FUNCTION_BLOCK Outfeed EXTENDS FB_PackML_BaseModule
VAR
	iOutfeedxis				   : I_BasicAxis;				  // For most axis and component commands
	iOutfeedAxisComponent	   : I_ComponentBase;			  // For registering the component with the EM
	iExternalSetpointGenerator : I_ExternalSetpointGenerator; // For setting properties of the External Setpoint Generator
END_VAR

// This method contains code which will execute when this PackML module is in the Aborting state
METHOD PROTECTED Aborting

// Note: The Abort command should be associated with the fault handing routine of a module. It should not be directly commanded from any user inteface. 

// This method is called as required by <c>StateControl()</c>
CASE SequenceState OF
	0:
		NoStateTasksToComplete := FALSE;
		SequenceState		   := SequenceState + 10;

	10:
		IF NOT iOutfeedxis.Error THEN
			IF iOutfeedxis.Stop() THEN
				SequenceState := SequenceState + 10;
			END_IF
		ELSE
			SequenceState := SequenceState + 10;
		END_IF

	20:
		IF iOutfeedxis.Stopped THEN
			SequenceState := SequenceState + 10;
		END_IF

	30:
		IF iOutfeedxis.Disable() THEN
			SequenceState := SequenceState + 10;
		END_IF

	40:
		IF NOT iOutfeedxis.Enabled THEN
			SequenceState := SequenceState + 10;
		END_IF

	50:
		StateTasksComplete := TRUE;
END_CASE

SUPER^.Aborting();
END_METHOD

// This method contains code which will execute when this PackML module is in the Clearing state
METHOD PROTECTED Clearing
VAR
	i				: UDINT;
	SubModulesReady : BOOL := TRUE;
END_VAR

// Note: The Clear command can also be thought of as a fault reset depite the ambiguity in the naming of the Reset state. 

// This method is called as required by <c>StateControl()</c>
CASE SequenceState OF
	0:
		NoStateTasksToComplete := FALSE;
		SequenceState		   := SequenceState + 10;

	10:
		IF iOutfeedxis.Reset() THEN
			SequenceState := SequenceState + 10;
		END_IF

	20:
		IF NOT iOutfeedxis.Error THEN
			SequenceState := SequenceState + 10;
		END_IF

	30:
		StateTasksComplete := TRUE;
END_CASE

SUPER^.Clearing();
END_METHOD

// This method contains code which will execute when this PackML module is in the Execute state
METHOD PROTECTED Execute
VAR
	

END_VAR

(*
The base implementation of this method is empty. User must override this method to provide functionality.
This method is called as required by StateControl()
*)
VAR
	Position : LREAL;
END_VAR
CASE _CurrentMode OF
	E_PMLUnitMode.ePMLUnitMode_Production:
		CASE SequenceState OF
			0:
				iExternalSetpointGenerator.Direction   := 1;
				iExternalSetpointGenerator.Destination := 0.0;
				iExternalSetpointGenerator.Velocity	   := 0.0;
				iExternalSetpointGenerator.Accel	   := 0.0;
				SequenceState						   := 10;

			10:
				IF iOutfeedxis.RunExternalSequence() THEN
					SequenceState := 20;
				END_IF

			20:
				IF iOutfeedxis.Axis.Status.HasJob THEN //Setpoint generator is operational
					SequenceState := 30;
				END_IF

			30: // Raise Velocity

				//ExtSetpointGen.Velocity := VelocityAxis.ActualVelocity + ((100.0 - VelocityAxis.ActualVelocity) * 0.01); // Without encoder feedback the Actual Velocity will stay at 0
				iExternalSetpointGenerator.Velocity := iExternalSetpointGenerator.Velocity + 0.01;
				IF iOutfeedxis.SetVelocity > 100.0 THEN
					SequenceState := 40;
				END_IF

			40: // Reduce Velocity to 0

				//ExtSetpointGen.Velocity := VelocityAxis.ActualVelocity - ((0.0 - VelocityAxis.ActualVelocity) * 0.01); // Without encoder feedback the Actual Velocity will stay at 0
				iExternalSetpointGenerator.Velocity := iExternalSetpointGenerator.Velocity - 0.01;
				IF (iExternalSetpointGenerator.Velocity <= 1.0) AND (iOutfeedxis.ActualVelocity = 0) THEN
					SequenceState := 50;
				END_IF

			50:
				IF iExternalSetpointGenerator.Disable() THEN
					SequenceState := 60;
				END_IF

			60:
				;
		END_CASE
END_CASE
END_METHOD

// Basic module initialization logic
METHOD PROTECTED Initialize : BOOL;
VAR
END_VAR

// This method is called by CyclicLogic() as required
Initialize := FALSE;
CASE DescendantSequenceState OF
	0:
		// Interfaces to connect to Components in the Fast_Task
		iOutfeedxis				   := Fast_Task.VelocityAxis;	   // For most axis and component commands
		iOutfeedAxisComponent	   := Fast_Task.VelocityAxis;	   // For registering the component with the EM
		iExternalSetpointGenerator := Fast_Task.VelExtSetpointGen; // For setting properties of the External Setpoint Generator

		//
		RegisterComponent(Component := iOutfeedAxisComponent);
		DescendantSequenceState := DescendantSequenceState + 10;

	10:
		IF SUPER^.Initialize() THEN
			DescendantSequenceState := DescendantSequenceState + 10;
		END_IF

	20:
		Initialize := TRUE;
END_CASE
END_METHOD

METHOD PROTECTED Resetting
VAR
END_VAR
CASE SequenceState OF
	0:
		NoStateTasksToComplete := FALSE;
		SequenceState		   := SequenceState + 10;

	10:
		IF iOutfeedxis.Enable() THEN
			SequenceState := SequenceState + 10;
		END_IF

	20:
		IF iOutfeedxis.Enabled THEN
			SequenceState := SequenceState + 10;
		END_IF

	30:
		StateTasksComplete := TRUE;
END_CASE

SUPER^.Resetting();
END_METHOD

END_FUNCTION_BLOCK

(* stored: Version 1.1.0.1, ProductVersion 3.1.4024.12
   POU Outfeed: Id {e948bf20-f0b6-46b0-a57a-2af964224def}, SpecialFunc None
   Method Aborting: Id {43b0d5d1-0b34-4df9-abc6-77c43e338e59}
   Method Clearing: Id {efefb995-793d-416a-9b69-702844c41757}
   Method Execute: Id {93af2509-69ae-4bef-9bf6-de48ad55d413}
   Method Initialize: Id {e3d83f98-ed74-4b99-8e16-5707372c199a}
   Method Resetting: Id {98759c75-0602-4f28-90ed-a645ad15f32d} *)
